FUNCTION_BLOCK FB_Module01 EXTENDS FB_Component
VAR_INPUT
	bPowerOn:				BOOL;
	bFuse1:					BOOL;
END_VAR
VAR_OUTPUT
END_VAR
VAR
	fbLogger:					FB_ListLogger;
	fbAlarm:					FB_Alarm;
	fbComponent1:				FB_Component;
	fbComponent2:				FB_Component;
	fbComponent3:				FB_Component;
	fbComponent4:				FB_ComponentEX;
END_VAR

SUPER^();

fbComponent1();
fbComponent2();
fbComponent3();
fbComponent4();

METHOD PROTECTED M_Active
VAR_INPUT
END_VAR
SUPER^.M_Active();

IF NOT bPowerOn THEN
	fbEvent.M_Add('Test');
	fbEvent.M_Add('Test2');
	fbEvent.M_Add('Test3');
	fbEvent.M_Error('Power not on', 2 ,E_Behaviour.Abort);
ELSIF NOT bFuse1 THEN
	fbEvent.M_Add('Test');
	fbEvent.M_Add('Test2');
	fbEvent.M_Add('Test3');
	fbEvent.M_Error('Fuse Triped', 3 ,E_Behaviour.Stop);	
	
END_IF
END_METHOD

METHOD PROTECTED M_Initialise : BOOL
VAR_INPUT
END_VAR
IF SUPER^.M_Initialise() THEN
	fbEvent.P_Logger:= fbLogger;
	fbLogger.M_Add(fbAlarm);

	fbSaftey.fbEvent.P_Logger:= fbLogger;
	fbSaftey.fbObserver.M_Attach(THIS^);


	fbComponent1.fbEvent.P_Logger:= fbLogger;
	fbComponent1.fbObserver.M_Attach(THIS^);
	fbObserver.M_Attach(fbComponent1);
	
	fbComponent2.fbEvent.P_Logger:= fbLogger;
	fbComponent2.fbObserver.M_Attach(THIS^);
	fbObserver.M_Attach(fbComponent2);
	
	fbComponent3.fbEvent.P_Logger:= fbLogger;
	fbComponent3.fbObserver.M_Attach(THIS^);
	fbObserver.M_Attach(fbComponent3);
	
	fbComponent4.fbEvent.P_Logger:= fbLogger;
	fbComponent4.fbObserver.M_Attach(THIS^);
	fbObserver.M_Attach(fbComponent4);
	M_Initialise:= TRUE;
END_IF
END_METHOD

METHOD PROTECTED M_Resetting : BOOL
VAR_INPUT
END_VAR
VAR
	nIndex:					DINT;
END_VAR
M_Resetting:= TRUE;
WHILE nIndex < fbObserver.nLength DO
	fbObserver.M_Index(nIndex).M_Request(E_Request.Reset);
	nIndex:= nIndex +1;
END_WHILE

fbAlarm.M_Reset();
END_METHOD

METHOD PROTECTED M_Starting : BOOL
VAR_INPUT
END_VAR
VAR
	nIndex:					DINT;
END_VAR
M_Starting:= TRUE;
WHILE nIndex < fbObserver.nLength DO
	M_Starting:= M_Starting AND fbObserver.M_Index(nIndex).M_Request(E_Request.Start);
	nIndex:= nIndex +1;
END_WHILE
END_METHOD

END_FUNCTION_BLOCK

(* stored: Version 1.1.0.1, ProductVersion 3.1.4024.12
   POU FB_Module01: Id {3744d03d-359c-4ab8-84fb-4ea93b7a5162}, SpecialFunc None
   Method M_Active: Id {eaffebca-5ff2-4f17-be84-3310a9ace22e}
   Method M_Initialise: Id {714c485c-83a6-4af2-a706-fec3f6b598e5}
   Method M_Resetting: Id {fa00b107-60e3-427f-9569-a0a34888482b}
   Method M_Starting: Id {12752945-7cd6-464f-965a-f81c0b828bfd} *)
